PROGRAM PRG_1
VAR
	bAlarm: BOOL;
	
	stMachine : ST_Machine;
END_VAR


stMachine.rTemperature := 85.0; 
stMachine.bRunning := TRUE;
bAlarm := F_CheckAlarm( stMachine);

 

 
IF F_IsOverheat(stMachine.rTemperature) THEN 
   stMachine.bRunning := FALSE; 
END_IF

END_PROGRAM

(* stored: Version 1.1.0.1, ProductVersion 3.1.4024.16
   POU PRG_1: Id {0fb5cfff-2da5-45df-8e63-305b0d4dc824}, SpecialFunc None *)
